DATA_BLOCK "T_HISTERESE"   // DB2
{ S7_Optimized_Access := 'TRUE' }
// stored: AutoNumber true, InstanceOfName IEC_TIMER, OfSystemLibElement IEC_TIMER, OfSystemLibVersion 1.0
"IEC_TIMER"
   // VAR
   //    PT : Time;
   //    ET { ExternalWritable := 'False'} : Time;
   //    IN : Bool;
   //    Q { ExternalWritable := 'False'} : Bool;
   // END_VAR
BEGIN
END_DATA_BLOCK

DATA_BLOCK "EncoderCh0-CarriageA"   // DB102
// stored: AutoNumber false, InstanceOfName CTRL_HSC, OfSystemLibElement CTRL_HSC, OfSystemLibVersion 1.0
"CTRL_HSC"
   // VAR_INPUT
   //    HSC : HW_HSC;
   //    DIR : Bool;
   //    CV : Bool;
   //    RV : Bool;
   //    PERIOD : Bool;
   //    NEW_DIR : Int;
   //    NEW_CV : DInt;
   //    NEW_RV : DInt;
   //    NEW_PERIOD : Int;
   // END_VAR
   // VAR_OUTPUT
   //    BUSY : Bool;
   //    STATUS : Word;
   // END_VAR
BEGIN
END_DATA_BLOCK

DATA_BLOCK "EncoderCh1-CarriageB"   // DB103
// stored: AutoNumber false, InstanceOfName CTRL_HSC, OfSystemLibElement CTRL_HSC, OfSystemLibVersion 1.0
"CTRL_HSC"
   // VAR_INPUT
   //    HSC : HW_HSC;
   //    DIR : Bool;
   //    CV : Bool;
   //    RV : Bool;
   //    PERIOD : Bool;
   //    NEW_DIR : Int;
   //    NEW_CV : DInt;
   //    NEW_RV : DInt;
   //    NEW_PERIOD : Int;
   // END_VAR
   // VAR_OUTPUT
   //    BUSY : Bool;
   //    STATUS : Word;
   // END_VAR
BEGIN
END_DATA_BLOCK

DATA_BLOCK "IEC_Timer_0_DB"   // DB15
{ S7_Optimized_Access := 'TRUE' }
// stored: AutoNumber true, InstanceOfName IEC_TIMER, OfSystemLibElement IEC_TIMER, OfSystemLibVersion 1.0
"IEC_TIMER"
   // VAR
   //    PT : Time;
   //    ET { ExternalWritable := 'False'} : Time;
   //    IN : Bool;
   //    Q { ExternalWritable := 'False'} : Bool;
   // END_VAR
BEGIN
END_DATA_BLOCK

DATA_BLOCK "CNT_CICLO_ALTERNANCIA_BOMBAS"   // DB12
{ S7_Optimized_Access := 'TRUE' }
// stored: AutoNumber true, InstanceOfName IEC_COUNTER, OfSystemLibElement IEC_COUNTER, OfSystemLibVersion 1.0
"IEC_COUNTER"
   // VAR RETAIN
   //    CU : Bool;
   //    CD : Bool;
   //    R : Bool;
   //    LD : Bool;
   //    QU : Bool;
   //    QD : Bool;
   //    PV : Int;
   //    CV : Int;
   // END_VAR
BEGIN
END_DATA_BLOCK

DATA_BLOCK "CNT_FUNC_B1"   // DB14
{ S7_Optimized_Access := 'TRUE' }
// stored: AutoNumber true, InstanceOfName IEC_COUNTER, OfSystemLibElement IEC_COUNTER, OfSystemLibVersion 1.0
"IEC_COUNTER"
   // VAR RETAIN
   //    CU : Bool;
   //    CD : Bool;
   //    R : Bool;
   //    LD : Bool;
   //    QU : Bool;
   //    QD : Bool;
   //    PV : Int;
   //    CV : Int;
   // END_VAR
BEGIN
END_DATA_BLOCK

DATA_BLOCK "CNT_FUNC_B2"   // DB37
{ S7_Optimized_Access := 'TRUE' }
// stored: AutoNumber true, InstanceOfName IEC_COUNTER, OfSystemLibElement IEC_COUNTER, OfSystemLibVersion 1.0
"IEC_COUNTER"
   // VAR RETAIN
   //    CU : Bool;
   //    CD : Bool;
   //    R : Bool;
   //    LD : Bool;
   //    QU : Bool;
   //    QD : Bool;
   //    PV : Int;
   //    CV : Int;
   // END_VAR
BEGIN
END_DATA_BLOCK

DATA_BLOCK "CNT_FUNC_B3"   // DB39
{ S7_Optimized_Access := 'TRUE' }
// stored: AutoNumber true, InstanceOfName IEC_COUNTER, OfSystemLibElement IEC_COUNTER, OfSystemLibVersion 1.0
"IEC_COUNTER"
   // VAR RETAIN
   //    CU : Bool;
   //    CD : Bool;
   //    R : Bool;
   //    LD : Bool;
   //    QU : Bool;
   //    QD : Bool;
   //    PV : Int;
   //    CV : Int;
   // END_VAR
BEGIN
END_DATA_BLOCK

DATA_BLOCK "Hold_Pulse"   // DB41
{ S7_Optimized_Access := 'TRUE' }
// stored: AutoNumber true, InstanceOfName IEC_TIMER, OfSystemLibElement IEC_TIMER, OfSystemLibVersion 1.0
"IEC_TIMER"
   // VAR
   //    PT : Time;
   //    ET { ExternalWritable := 'False'} : Time;
   //    IN : Bool;
   //    Q { ExternalWritable := 'False'} : Bool;
   // END_VAR
BEGIN
END_DATA_BLOCK

DATA_BLOCK "PERÍODO_ALTERNANCIA_BOMBAS"   // DB10
{ S7_Optimized_Access := 'TRUE' }
// stored: AutoNumber true, InstanceOfName IEC_TIMER, OfSystemLibElement IEC_TIMER, OfSystemLibVersion 1.0
"IEC_TIMER"
   // VAR RETAIN
   //    PT : Time;
   //    ET { ExternalWritable := 'False'} : Time;
   //    IN : Bool;
   //    Q { ExternalWritable := 'False'} : Bool;
   // END_VAR
BEGIN
END_DATA_BLOCK

DATA_BLOCK "TEMP_FUNC_B1"   // DB13
{ S7_Optimized_Access := 'TRUE' }
// stored: AutoNumber true, InstanceOfName IEC_TIMER, OfSystemLibElement IEC_TIMER, OfSystemLibVersion 1.0
"IEC_TIMER"
   // VAR
   //    PT : Time;
   //    ET { ExternalWritable := 'False'} : Time;
   //    IN : Bool;
   //    Q { ExternalWritable := 'False'} : Bool;
   // END_VAR
BEGIN
END_DATA_BLOCK

DATA_BLOCK "TEMP_FUNC_B2"   // DB15
{ S7_Optimized_Access := 'TRUE' }
// stored: AutoNumber true, InstanceOfName IEC_TIMER, OfSystemLibElement IEC_TIMER, OfSystemLibVersion 1.0
"IEC_TIMER"
   // VAR
   //    PT : Time;
   //    ET { ExternalWritable := 'False'} : Time;
   //    IN : Bool;
   //    Q { ExternalWritable := 'False'} : Bool;
   // END_VAR
BEGIN
END_DATA_BLOCK

DATA_BLOCK "TEMP_FUNC_B3"   // DB38
{ S7_Optimized_Access := 'TRUE' }
// stored: AutoNumber true, InstanceOfName IEC_TIMER, OfSystemLibElement IEC_TIMER, OfSystemLibVersion 1.0
"IEC_TIMER"
   // VAR
   //    PT : Time;
   //    ET { ExternalWritable := 'False'} : Time;
   //    IN : Bool;
   //    Q { ExternalWritable := 'False'} : Bool;
   // END_VAR
BEGIN
END_DATA_BLOCK

DATA_BLOCK "T_ABERTURA_EV1.1_HMI"   // DB16
{ S7_Optimized_Access := 'TRUE' }
// stored: AutoNumber true, InstanceOfName IEC_TIMER, OfSystemLibElement IEC_TIMER, OfSystemLibVersion 1.0
"IEC_TIMER"
   // VAR
   //    PT : Time;
   //    ET { ExternalWritable := 'False'} : Time;
   //    IN : Bool;
   //    Q { ExternalWritable := 'False'} : Bool;
   // END_VAR
BEGIN
END_DATA_BLOCK

DATA_BLOCK "T_ABERTURA_EV1.2_HMI"   // DB27
{ S7_Optimized_Access := 'TRUE' }
// stored: AutoNumber true, InstanceOfName IEC_TIMER, OfSystemLibElement IEC_TIMER, OfSystemLibVersion 1.0
"IEC_TIMER"
   // VAR
   //    PT : Time;
   //    ET { ExternalWritable := 'False'} : Time;
   //    IN : Bool;
   //    Q { ExternalWritable := 'False'} : Bool;
   // END_VAR
BEGIN
END_DATA_BLOCK

DATA_BLOCK "T_ABERTURA_EV2.1_HMI"   // DB19
{ S7_Optimized_Access := 'TRUE' }
// stored: AutoNumber true, InstanceOfName IEC_TIMER, OfSystemLibElement IEC_TIMER, OfSystemLibVersion 1.0
"IEC_TIMER"
   // VAR
   //    PT : Time;
   //    ET { ExternalWritable := 'False'} : Time;
   //    IN : Bool;
   //    Q { ExternalWritable := 'False'} : Bool;
   // END_VAR
BEGIN
END_DATA_BLOCK

DATA_BLOCK "T_ABERTURA_EV2.2_HMI"   // DB29
{ S7_Optimized_Access := 'TRUE' }
// stored: AutoNumber true, InstanceOfName IEC_TIMER, OfSystemLibElement IEC_TIMER, OfSystemLibVersion 1.0
"IEC_TIMER"
   // VAR
   //    PT : Time;
   //    ET { ExternalWritable := 'False'} : Time;
   //    IN : Bool;
   //    Q { ExternalWritable := 'False'} : Bool;
   // END_VAR
BEGIN
END_DATA_BLOCK

DATA_BLOCK "T_ABERTURA_EV3.1_HMI"   // DB21
{ S7_Optimized_Access := 'TRUE' }
// stored: AutoNumber true, InstanceOfName IEC_TIMER, OfSystemLibElement IEC_TIMER, OfSystemLibVersion 1.0
"IEC_TIMER"
   // VAR
   //    PT : Time;
   //    ET { ExternalWritable := 'False'} : Time;
   //    IN : Bool;
   //    Q { ExternalWritable := 'False'} : Bool;
   // END_VAR
BEGIN
END_DATA_BLOCK

DATA_BLOCK "T_ABERTURA_EV3.2_HMI"   // DB31
{ S7_Optimized_Access := 'TRUE' }
// stored: AutoNumber true, InstanceOfName IEC_TIMER, OfSystemLibElement IEC_TIMER, OfSystemLibVersion 1.0
"IEC_TIMER"
   // VAR
   //    PT : Time;
   //    ET { ExternalWritable := 'False'} : Time;
   //    IN : Bool;
   //    Q { ExternalWritable := 'False'} : Bool;
   // END_VAR
BEGIN
END_DATA_BLOCK

DATA_BLOCK "T_ABERTURA_EV4.1_HMI"   // DB23
{ S7_Optimized_Access := 'TRUE' }
// stored: AutoNumber true, InstanceOfName IEC_TIMER, OfSystemLibElement IEC_TIMER, OfSystemLibVersion 1.0
"IEC_TIMER"
   // VAR
   //    PT : Time;
   //    ET { ExternalWritable := 'False'} : Time;
   //    IN : Bool;
   //    Q { ExternalWritable := 'False'} : Bool;
   // END_VAR
BEGIN
END_DATA_BLOCK

DATA_BLOCK "T_ABERTURA_EV4.2_HMI"   // DB33
{ S7_Optimized_Access := 'TRUE' }
// stored: AutoNumber true, InstanceOfName IEC_TIMER, OfSystemLibElement IEC_TIMER, OfSystemLibVersion 1.0
"IEC_TIMER"
   // VAR
   //    PT : Time;
   //    ET { ExternalWritable := 'False'} : Time;
   //    IN : Bool;
   //    Q { ExternalWritable := 'False'} : Bool;
   // END_VAR
BEGIN
END_DATA_BLOCK

DATA_BLOCK "T_ABERTURA_EV5.1_HMI"   // DB25
{ S7_Optimized_Access := 'TRUE' }
// stored: AutoNumber true, InstanceOfName IEC_TIMER, OfSystemLibElement IEC_TIMER, OfSystemLibVersion 1.0
"IEC_TIMER"
   // VAR
   //    PT : Time;
   //    ET { ExternalWritable := 'False'} : Time;
   //    IN : Bool;
   //    Q { ExternalWritable := 'False'} : Bool;
   // END_VAR
BEGIN
END_DATA_BLOCK

DATA_BLOCK "T_ABERTURA_EV5.2_HMI"   // DB35
{ S7_Optimized_Access := 'TRUE' }
// stored: AutoNumber true, InstanceOfName IEC_TIMER, OfSystemLibElement IEC_TIMER, OfSystemLibVersion 1.0
"IEC_TIMER"
   // VAR
   //    PT : Time;
   //    ET { ExternalWritable := 'False'} : Time;
   //    IN : Bool;
   //    Q { ExternalWritable := 'False'} : Bool;
   // END_VAR
BEGIN
END_DATA_BLOCK

DATA_BLOCK "T_FECHO_EV1.1_HMI"   // DB17
{ S7_Optimized_Access := 'TRUE' }
// stored: AutoNumber true, InstanceOfName IEC_TIMER, OfSystemLibElement IEC_TIMER, OfSystemLibVersion 1.0
"IEC_TIMER"
   // VAR
   //    PT : Time;
   //    ET { ExternalWritable := 'False'} : Time;
   //    IN : Bool;
   //    Q { ExternalWritable := 'False'} : Bool;
   // END_VAR
BEGIN
END_DATA_BLOCK

DATA_BLOCK "T_FECHO_EV1.2_HMI"   // DB28
{ S7_Optimized_Access := 'TRUE' }
// stored: AutoNumber true, InstanceOfName IEC_TIMER, OfSystemLibElement IEC_TIMER, OfSystemLibVersion 1.0
"IEC_TIMER"
   // VAR
   //    PT : Time;
   //    ET { ExternalWritable := 'False'} : Time;
   //    IN : Bool;
   //    Q { ExternalWritable := 'False'} : Bool;
   // END_VAR
BEGIN
END_DATA_BLOCK

DATA_BLOCK "T_FECHO_EV2.1_HMI"   // DB20
{ S7_Optimized_Access := 'TRUE' }
// stored: AutoNumber true, InstanceOfName IEC_TIMER, OfSystemLibElement IEC_TIMER, OfSystemLibVersion 1.0
"IEC_TIMER"
   // VAR
   //    PT : Time;
   //    ET { ExternalWritable := 'False'} : Time;
   //    IN : Bool;
   //    Q { ExternalWritable := 'False'} : Bool;
   // END_VAR
BEGIN
END_DATA_BLOCK

DATA_BLOCK "T_FECHO_EV2.2_HMI"   // DB30
{ S7_Optimized_Access := 'TRUE' }
// stored: AutoNumber true, InstanceOfName IEC_TIMER, OfSystemLibElement IEC_TIMER, OfSystemLibVersion 1.0
"IEC_TIMER"
   // VAR
   //    PT : Time;
   //    ET { ExternalWritable := 'False'} : Time;
   //    IN : Bool;
   //    Q { ExternalWritable := 'False'} : Bool;
   // END_VAR
BEGIN
END_DATA_BLOCK

DATA_BLOCK "T_FECHO_EV3.1_HMI"   // DB22
{ S7_Optimized_Access := 'TRUE' }
// stored: AutoNumber true, InstanceOfName IEC_TIMER, OfSystemLibElement IEC_TIMER, OfSystemLibVersion 1.0
"IEC_TIMER"
   // VAR
   //    PT : Time;
   //    ET { ExternalWritable := 'False'} : Time;
   //    IN : Bool;
   //    Q { ExternalWritable := 'False'} : Bool;
   // END_VAR
BEGIN
END_DATA_BLOCK

DATA_BLOCK "T_FECHO_EV3.2_HMI"   // DB32
{ S7_Optimized_Access := 'TRUE' }
// stored: AutoNumber true, InstanceOfName IEC_TIMER, OfSystemLibElement IEC_TIMER, OfSystemLibVersion 1.0
"IEC_TIMER"
   // VAR
   //    PT : Time;
   //    ET { ExternalWritable := 'False'} : Time;
   //    IN : Bool;
   //    Q { ExternalWritable := 'False'} : Bool;
   // END_VAR
BEGIN
END_DATA_BLOCK

DATA_BLOCK "T_FECHO_EV4.1_HMI"   // DB24
{ S7_Optimized_Access := 'TRUE' }
// stored: AutoNumber true, InstanceOfName IEC_TIMER, OfSystemLibElement IEC_TIMER, OfSystemLibVersion 1.0
"IEC_TIMER"
   // VAR
   //    PT : Time;
   //    ET { ExternalWritable := 'False'} : Time;
   //    IN : Bool;
   //    Q { ExternalWritable := 'False'} : Bool;
   // END_VAR
BEGIN
END_DATA_BLOCK

DATA_BLOCK "T_FECHO_EV4.2_HMI"   // DB34
{ S7_Optimized_Access := 'TRUE' }
// stored: AutoNumber true, InstanceOfName IEC_TIMER, OfSystemLibElement IEC_TIMER, OfSystemLibVersion 1.0
"IEC_TIMER"
   // VAR
   //    PT : Time;
   //    ET { ExternalWritable := 'False'} : Time;
   //    IN : Bool;
   //    Q { ExternalWritable := 'False'} : Bool;
   // END_VAR
BEGIN
END_DATA_BLOCK

DATA_BLOCK "T_FECHO_EV5.1_HMI"   // DB26
{ S7_Optimized_Access := 'TRUE' }
// stored: AutoNumber true, InstanceOfName IEC_TIMER, OfSystemLibElement IEC_TIMER, OfSystemLibVersion 1.0
"IEC_TIMER"
   // VAR
   //    PT : Time;
   //    ET { ExternalWritable := 'False'} : Time;
   //    IN : Bool;
   //    Q { ExternalWritable := 'False'} : Bool;
   // END_VAR
BEGIN
END_DATA_BLOCK

DATA_BLOCK "T_FECHO_EV5.2_HMI"   // DB36
{ S7_Optimized_Access := 'TRUE' }
// stored: AutoNumber true, InstanceOfName IEC_TIMER, OfSystemLibElement IEC_TIMER, OfSystemLibVersion 1.0
"IEC_TIMER"
   // VAR
   //    PT : Time;
   //    ET { ExternalWritable := 'False'} : Time;
   //    IN : Bool;
   //    Q { ExternalWritable := 'False'} : Bool;
   // END_VAR
BEGIN
END_DATA_BLOCK

DATA_BLOCK "T_LAVAGEM"   // DB4
{ S7_Optimized_Access := 'TRUE' }
// stored: AutoNumber true, InstanceOfName IEC_TIMER, OfSystemLibElement IEC_TIMER, OfSystemLibVersion 1.0
"IEC_TIMER"
   // VAR RETAIN
   //    PT : Time;
   //    ET { ExternalWritable := 'False'} : Time;
   //    IN : Bool;
   //    Q { ExternalWritable := 'False'} : Bool;
   // END_VAR
BEGIN
END_DATA_BLOCK

DATA_BLOCK "T_POS_EVS"   // DB3
{ S7_Optimized_Access := 'TRUE' }
// stored: AutoNumber true, InstanceOfName IEC_TIMER, OfSystemLibElement IEC_TIMER, OfSystemLibVersion 1.0
"IEC_TIMER"
   // VAR
   //    PT : Time;
   //    ET { ExternalWritable := 'False'} : Time;
   //    IN : Bool;
   //    Q { ExternalWritable := 'False'} : Bool;
   // END_VAR
BEGIN
END_DATA_BLOCK

DATA_BLOCK "T_PRESS_FILT_1"   // DB8
{ S7_Optimized_Access := 'TRUE' }
// stored: AutoNumber true, InstanceOfName IEC_TIMER, OfSystemLibElement IEC_TIMER, OfSystemLibVersion 1.0
"IEC_TIMER"
   // VAR
   //    PT : Time;
   //    ET { ExternalWritable := 'False'} : Time;
   //    IN : Bool;
   //    Q { ExternalWritable := 'False'} : Bool;
   // END_VAR
BEGIN
END_DATA_BLOCK

DATA_BLOCK "T_PRESS_FILT_2"   // DB9
{ S7_Optimized_Access := 'TRUE' }
// stored: AutoNumber true, InstanceOfName IEC_TIMER, OfSystemLibElement IEC_TIMER, OfSystemLibVersion 1.0
"IEC_TIMER"
   // VAR
   //    PT : Time;
   //    ET { ExternalWritable := 'False'} : Time;
   //    IN : Bool;
   //    Q { ExternalWritable := 'False'} : Bool;
   // END_VAR
BEGIN
END_DATA_BLOCK

DATA_BLOCK "T_RINSE"   // DB5
{ S7_Optimized_Access := 'TRUE' }
// stored: AutoNumber true, InstanceOfName IEC_TIMER, OfSystemLibElement IEC_TIMER, OfSystemLibVersion 1.0
"IEC_TIMER"
   // VAR RETAIN
   //    PT : Time;
   //    ET { ExternalWritable := 'False'} : Time;
   //    IN : Bool;
   //    Q { ExternalWritable := 'False'} : Bool;
   // END_VAR
BEGIN
END_DATA_BLOCK

DATA_BLOCK "T_STOP_BOMBAS"   // DB2
{ S7_Optimized_Access := 'TRUE' }
// stored: AutoNumber true, InstanceOfName IEC_TIMER, OfSystemLibElement IEC_TIMER, OfSystemLibVersion 1.0
"IEC_TIMER"
   // VAR
   //    PT : Time;
   //    ET { ExternalWritable := 'False'} : Time;
   //    IN : Bool;
   //    Q { ExternalWritable := 'False'} : Bool;
   // END_VAR
BEGIN
END_DATA_BLOCK
